INTERFACE I_ResponseIdGenerator

METHOD PUBLIC Generate : T_MAXSTRING
VAR_INPUT
END_VAR
END_METHOD

END_INTERFACE

(* stored: Version 1.1.0.1, ProductVersion 3.1.4024.12
   Itf I_ResponseIdGenerator: Id {a3a52b48-80d7-0738-0a64-e09497b0074b}
   Method Generate: Id {844835a0-bc52-08f6-3590-ccb12681aaa7} *)
